(* IEC 61131-3 sources: vytah_teco/, 10 files *)

(* ---- VYTAH_TECO.ST ---- *)
TYPE
  TUsintArray : ARRAY [1..5] OF USINT;
END_TYPE

VAR_GLOBAL
  init : BOOL := 1;                                 //inicializace
  otvp : BOOL := 0;                                 //otevirani pravych dveri
  otvl : BOOL := 0;                                 //          levych
  kp : USINT := 1;                                  //poloha prave kabiny
  kl : USINT := 1;                                  //       leve
  kamp : USINT := 0;                                //kam ma prava kabina prijet
  kaml : USINT := 0;                                //       leva
  i : USINT;                                        //na PWM
  prava : TUsintArray := [0,0,0,0,0];               //pozadavky na pravou kabinu
  leva : TUsintArray := [0,0,0,0,0];                //             levou
  dol : ARRAY[1..5] OF BOOL := [0,0,0,0,0];
  nah : ARRAY[1..5] OF BOOL := [0,0,0,0,0];
END_VAR

(* ---- fceIn.ST ---- *)
FUNCTION fceIn : BOOL
  VAR_INPUT
    p : USINT;
  END_VAR
  VAR_IN_OUT
    pole : TUsintArray;
  END_VAR
  VAR
    i : USINT;
  END_VAR
  VAR_TEMP
  END_VAR

  fceIn := 0;

  //if p = kaml then
    //fceIn := 1;
  //else
   for i := 1 to 5 do
    if p = pole[i] then fceIn := 1; end_if;
   end_for;
  //end_if;

END_FUNCTION

(* ---- fceMax.ST ---- *)
FUNCTION fceMax : USINT
  VAR_INPUT
  END_VAR
  VAR_IN_OUT
    pole : TUsintArray;
  END_VAR
  VAR
    i : USINT;
    m : USINT;
  END_VAR
  VAR_TEMP
  END_VAR

  m := 0;

  for i := 1 to 5 do
    if pole[i] > m then m := pole[i]; end_if;
  end_for;

  fceMax := m;

END_FUNCTION

(* ---- fceMin.ST ---- *)
FUNCTION fceMin : USINT
  VAR_INPUT
  END_VAR
  VAR_IN_OUT
    pole : TUsintArray;
  END_VAR
  VAR
    i : USINT;
    m : USINT;
  END_VAR
  VAR_TEMP
  END_VAR

  m := 6;

  for i := 1 to 5 do
    if pole[i] <> 0 and pole[i] < m then m := pole[i]; end_if;
  end_for;

  if m = 6 then m := 0; end_if;

  fceMin := m;

END_FUNCTION

(* ---- funkcePWM.ST ---- *)
FUNCTION funkcePWM : BOOL
  VAR_INPUT
    strida : USINT;
  END_VAR
  VAR_IN_OUT
  END_VAR
  VAR
    motor : BOOL;
  END_VAR
  VAR_TEMP

  END_VAR

  if strida>10 then strida:=10;
  end_if;

  motor:=0;
  if i<=strida then motor:=1;

  end_if;

  i:=i+1;

  if i>10 then i:=0;
  end_if;

  fcePWM:=motor;

END_FUNCTION

(* ---- fbDvere.ST ---- *)
FUNCTION_BLOCK fbDvere
  VAR_INPUT
  END_VAR
  VAR_OUTPUT
  END_VAR
  VAR_IN_OUT
  END_VAR
  VAR
    casovacl : TON;      //casovac levych dveri
    startl : BOOL;
    outputl : BOOL;
    casovacp : TON;      //casovac pravych dveri
    startp : BOOL;
    outputp : BOOL;
  END_VAR
  VAR_TEMP
  END_VAR

  if otvl then        //leve dvere
    casovacl( IN := startl, PT :=T#10s, Q => outputl );
    startl := 1;
    if pod1l then dvere1l := 1;          //vyber dveri v patre kabiny
    elsif pod2l then dvere2l := 1;
    elsif pod3l then dvere3l := 1;
    elsif pod4l then dvere4l := 1;
    elsif pod5l then dvere5l := 1;
    else otvl := 0; end_if;
    if casovacl.ET>T#5s then
        dvere1l := 0;
        dvere2l := 0;
        dvere3l := 0;
        dvere4l := 0;
        dvere5l := 0;
    end_if;
    if outputl then
        startl := 0;
        otvl := 0;
    end_if;
  end_if;

  if otvp then             //prave dvere
    casovacp( IN := startp, PT :=T#10s, Q => outputp );
    startp := 1;
    if pod1p then dvere1p := 1;         //vyber dveri v patre kabiny
    elsif pod2p then dvere2p := 1;
    elsif pod3p then dvere3p := 1;
    elsif pod4p then dvere4p := 1;
    elsif pod5p then dvere5p := 1;
    else otvp := 0; end_if;
    if casovacp.ET>T#5s then
        dvere1p := 0;
        dvere2p := 0;
        dvere3p := 0;
        dvere4p := 0;
        dvere5p := 0;
    end_if;
    if outputp then
        startp := 0;
        otvp := 0;
    end_if;
  end_if;

END_FUNCTION_BLOCK

(* ---- fbKabinal.ST ---- *)
FUNCTION_BLOCK fbKabinal
  VAR_INPUT
  END_VAR
  VAR_OUTPUT
  END_VAR
  VAR_IN_OUT
  END_VAR
  VAR
    vyjmout : fbVyjmout;
    st : USINT;
    m : BOOL := 0;
  END_VAR
  VAR_TEMP
  END_VAR

  if motor2A or motor1A then                                 //zmena aktualni hodnotz
    if pod1l then kl := 1;
    elsif pod2l then kl := 2;
    elsif pod3l then kl := 3;
    elsif pod4l then kl := 4;
    elsif pod5l then kl := 5;
    end_if;
  end_if;

    st := 10;
    if kl - kaml = 1 or kaml - kl = 1 then
      st := 7;
      if mezipL then
        m := 1;
      end_if;
      if m then
        st := 4;
      end_if;
    end_if;

    motor2A := 0;
    motor1A := 0;

 if kaml = kl then                                    //ovladani motoru
   otvl := 1;
   vyjmout(pole := leva);
   m := 0;
 elsif kaml <> 0 and not otvl then
  if kaml > kl then
    motor2A := funkcePWM(st);
  elsif kaml < kl then
    motor1A := funkcePWM(st);
  end_if;
 end_if;

END_FUNCTION_BLOCK

(* ---- fbKabinap.ST ---- *)
FUNCTION_BLOCK fbKabinap
  VAR_INPUT
  END_VAR
  VAR_OUTPUT
  END_VAR
  VAR_IN_OUT
  END_VAR
  VAR
    vyjmout : fbVyjmout;
    st : USINT;
    m : BOOL := 0;
  END_VAR
  VAR_TEMP
  END_VAR

  if motor4A or motor3A then                            //zmena aktualni hodnoty
    if pod1p then kp := 1;
    elsif pod2p then kp := 2;
    elsif pod3p then kp := 3;
    elsif pod4p then kp := 4;
    elsif pod5p then kp := 5;
    end_if;
  end_if;

    st := 10;
    if kp - kamp = 1 or kamp - kp = 1 then
      st := 7;
      if mezipP then
        m := 1;
      end_if;
      if m then
        st := 4;
      end_if;
    end_if;

    motor4A := 0;
    motor3A := 0;

 if kamp = kp then                             //ovladani motoru
   otvp := 1;
   vyjmout(pole := prava);
   m := 0;
 elsif kamp <> 0 and not otvp then
  if kamp > kp then
    motor4A := funkcePWM(st);
  elsif kamp < kp then
    motor3A := funkcePWM(st);
  end_if;
 end_if;

END_FUNCTION_BLOCK

(* ---- fbVyjmout.ST ---- *)
FUNCTION_BLOCK fbVyjmout
  VAR_INPUT
  END_VAR
  VAR_OUTPUT
  END_VAR
  VAR_IN_OUT
    pole : TUsintArray;
  END_VAR
  VAR
    i : USINT;
  END_VAR
  VAR_TEMP
  END_VAR

  //kaml := pole[1];
  for i := 1 to 4 do
    pole[i] := pole[i+1];
  end_for;
  pole[5] := 0;

END_FUNCTION_BLOCK

(* ---- prgMain.ST ---- *)
PROGRAM prgMain
  VAR_INPUT
  END_VAR
  VAR_OUTPUT
  END_VAR
  VAR

  END_VAR
  VAR_TEMP
  END_VAR
  (*ddddd*)

  (*mara*)

  (*ddddd*)
  (*ddddd*)

END_PROGRAM
